// TIA Portal V19 export
FUNCTION "SCALING_PARAMETERS" : Void   // FC4, LAD
{ S7_Optimized_Access := 'TRUE' }
// stored: SetENOAutomatically false
BEGIN

REGION Network 1: PH_SCALE
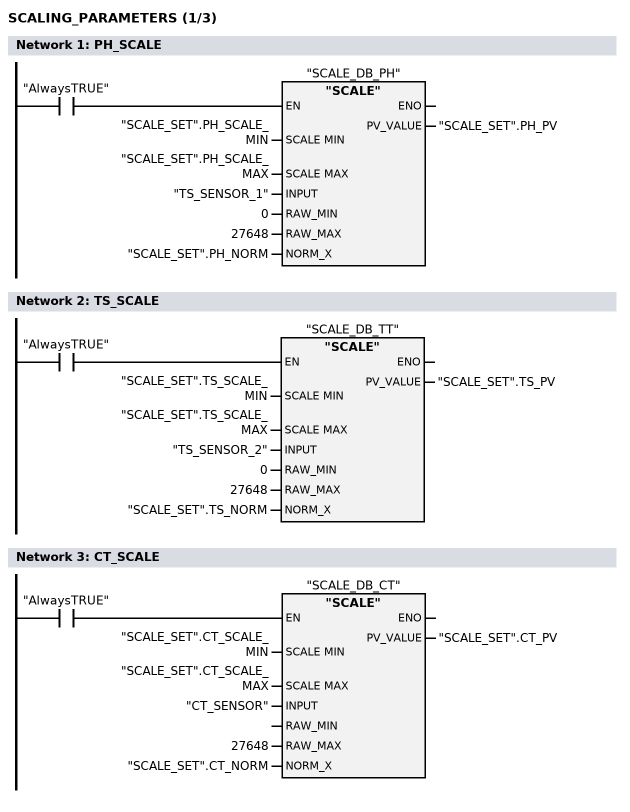
   RUNG wire#powerrail
      Contact( "AlwaysTRUE" )
      "SCALE_DB_PH"("SCALE MIN" := "SCALE_SET".PH_SCALE_MIN, "SCALE MAX" := "SCALE_SET".PH_SCALE_MAX, INPUT := "TS_SENSOR_1", RAW_MIN := 0, RAW_MAX := 27648, NORM_X := "SCALE_SET".PH_NORM, PV_VALUE => "SCALE_SET".PH_PV)
   END_RUNG
   // the same network as SCL:
   IF "AlwaysTRUE" THEN
       "SCALE_DB_PH"("SCALE MIN" := "SCALE_SET".PH_SCALE_MIN,   // "SCALE"
                     "SCALE MAX" := "SCALE_SET".PH_SCALE_MAX,
                     INPUT := "TS_SENSOR_1",
                     RAW_MIN := 0,
                     RAW_MAX := 27648,
                     NORM_X := "SCALE_SET".PH_NORM,
                     PV_VALUE => "SCALE_SET".PH_PV);
   END_IF;
END_REGION

REGION Network 2: TS_SCALE
   RUNG wire#powerrail
      Contact( "AlwaysTRUE" )
      "SCALE_DB_TT"("SCALE MIN" := "SCALE_SET".TS_SCALE_MIN, "SCALE MAX" := "SCALE_SET".TS_SCALE_MAX, INPUT := "TS_SENSOR_2", RAW_MIN := 0, RAW_MAX := 27648, NORM_X := "SCALE_SET".TS_NORM, PV_VALUE => "SCALE_SET".TS_PV)
   END_RUNG
   // the same network as SCL:
   IF "AlwaysTRUE" THEN
       "SCALE_DB_TT"("SCALE MIN" := "SCALE_SET".TS_SCALE_MIN,   // "SCALE"
                     "SCALE MAX" := "SCALE_SET".TS_SCALE_MAX,
                     INPUT := "TS_SENSOR_2",
                     RAW_MIN := 0,
                     RAW_MAX := 27648,
                     NORM_X := "SCALE_SET".TS_NORM,
                     PV_VALUE => "SCALE_SET".TS_PV);
   END_IF;
END_REGION

REGION Network 3: CT_SCALE
   RUNG wire#powerrail
      Contact( "AlwaysTRUE" )
      "SCALE_DB_CT"("SCALE MIN" := "SCALE_SET".CT_SCALE_MIN, "SCALE MAX" := "SCALE_SET".CT_SCALE_MAX, INPUT := "CT_SENSOR", RAW_MIN :=, RAW_MAX := 27648, NORM_X := "SCALE_SET".CT_NORM, PV_VALUE => "SCALE_SET".CT_PV)
   END_RUNG
   // the same network as SCL:
   IF "AlwaysTRUE" THEN
       "SCALE_DB_CT"("SCALE MIN" := "SCALE_SET".CT_SCALE_MIN,   // "SCALE"
                     "SCALE MAX" := "SCALE_SET".CT_SCALE_MAX,
                     INPUT := "CT_SENSOR",
                     RAW_MAX := 27648,
                     NORM_X := "SCALE_SET".CT_NORM,
                     PV_VALUE => "SCALE_SET".CT_PV);
   END_IF;
END_REGION

REGION Network 4: SET_PUMP_SPEED
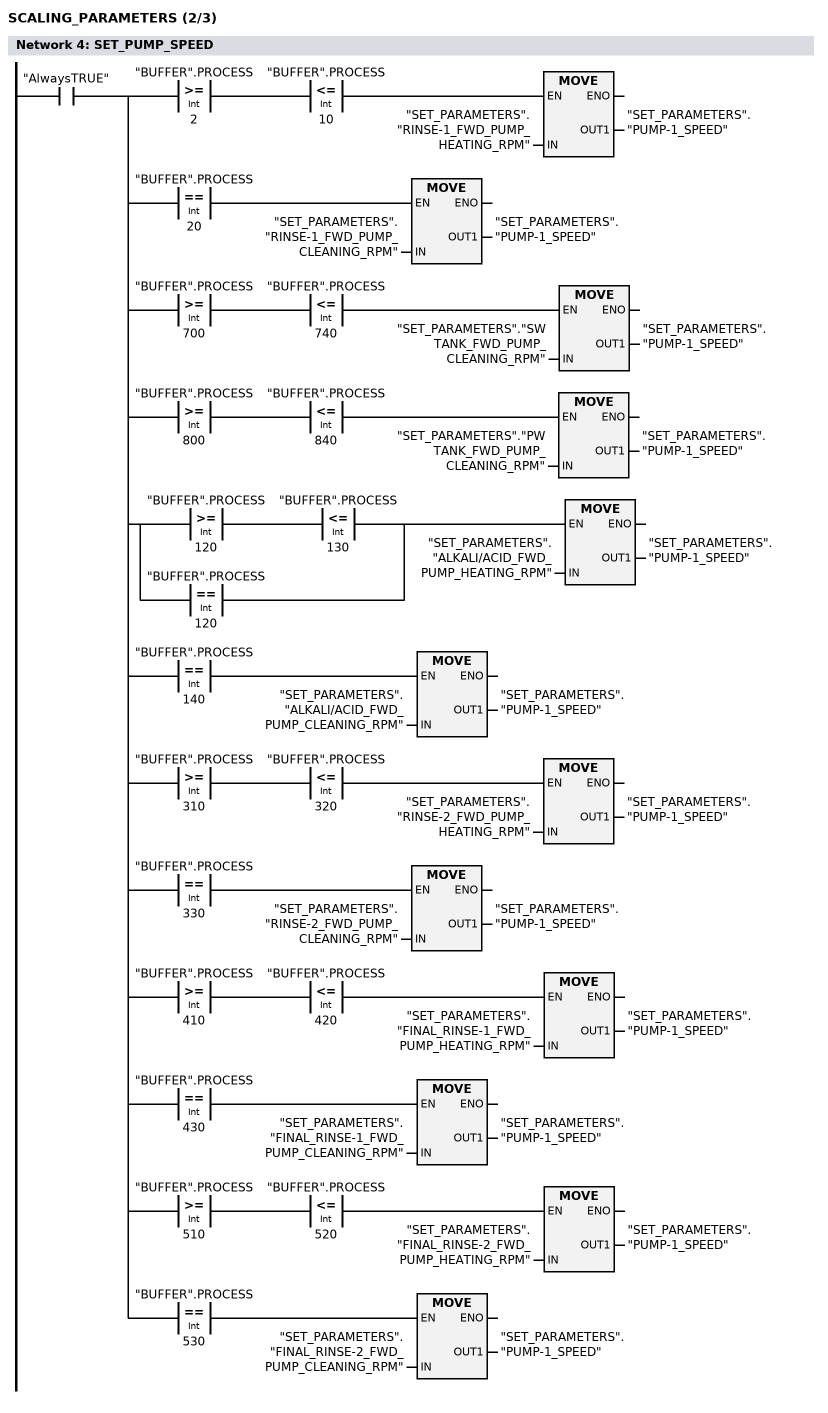
   RUNG wire#powerrail
      Contact( "AlwaysTRUE" )
      wire#w1
      { S7_Templates := "SrcType := Int" } GE_Contact(in1 := "BUFFER".PROCESS, in2 := 2)
      { S7_Templates := "SrcType := Int" } LE_Contact(in1 := "BUFFER".PROCESS, in2 := 10)
      Move(in := "SET_PARAMETERS"."RINSE-1_FWD_PUMP_HEATING_RPM", out1 => "SET_PARAMETERS"."PUMP-1_SPEED")
   END_RUNG
   RUNG wire#w1
      { S7_Templates := "SrcType := Int" } EQ_Contact(in1 := "BUFFER".PROCESS, in2 := 20)
      Move(in := "SET_PARAMETERS"."RINSE-1_FWD_PUMP_CLEANING_RPM", out1 => "SET_PARAMETERS"."PUMP-1_SPEED")
   END_RUNG
   RUNG wire#w1
      { S7_Templates := "SrcType := Int" } GE_Contact(in1 := "BUFFER".PROCESS, in2 := 700)
      { S7_Templates := "SrcType := Int" } LE_Contact(in1 := "BUFFER".PROCESS, in2 := 740)
      Move(in := "SET_PARAMETERS"."SW TANK_FWD_PUMP_CLEANING_RPM", out1 => "SET_PARAMETERS"."PUMP-1_SPEED")
   END_RUNG
   RUNG wire#w1
      { S7_Templates := "SrcType := Int" } GE_Contact(in1 := "BUFFER".PROCESS, in2 := 800)
      { S7_Templates := "SrcType := Int" } LE_Contact(in1 := "BUFFER".PROCESS, in2 := 840)
      Move(in := "SET_PARAMETERS"."PW TANK_FWD_PUMP_CLEANING_RPM", out1 => "SET_PARAMETERS"."PUMP-1_SPEED")
   END_RUNG
   RUNG wire#w1
      { S7_Templates := "SrcType := Int" } GE_Contact(in1 := "BUFFER".PROCESS, in2 := 120)
      { S7_Templates := "SrcType := Int" } LE_Contact(in1 := "BUFFER".PROCESS, in2 := 130)
      wire#w2
      Move(in := "SET_PARAMETERS"."ALKALI/ACID_FWD_PUMP_HEATING_RPM", out1 => "SET_PARAMETERS"."PUMP-1_SPEED")
   END_RUNG
   RUNG wire#w1
      { S7_Templates := "SrcType := Int" } EQ_Contact(in1 := "BUFFER".PROCESS, in2 := 120)
   END_RUNG wire#w2
   RUNG wire#w1
      { S7_Templates := "SrcType := Int" } EQ_Contact(in1 := "BUFFER".PROCESS, in2 := 140)
      Move(in := "SET_PARAMETERS"."ALKALI/ACID_FWD_PUMP_CLEANING_RPM", out1 => "SET_PARAMETERS"."PUMP-1_SPEED")
   END_RUNG
   RUNG wire#w1
      { S7_Templates := "SrcType := Int" } GE_Contact(in1 := "BUFFER".PROCESS, in2 := 310)
      { S7_Templates := "SrcType := Int" } LE_Contact(in1 := "BUFFER".PROCESS, in2 := 320)
      Move(in := "SET_PARAMETERS"."RINSE-2_FWD_PUMP_HEATING_RPM", out1 => "SET_PARAMETERS"."PUMP-1_SPEED")
   END_RUNG
   RUNG wire#w1
      { S7_Templates := "SrcType := Int" } EQ_Contact(in1 := "BUFFER".PROCESS, in2 := 330)
      Move(in := "SET_PARAMETERS"."RINSE-2_FWD_PUMP_CLEANING_RPM", out1 => "SET_PARAMETERS"."PUMP-1_SPEED")
   END_RUNG
   RUNG wire#w1
      { S7_Templates := "SrcType := Int" } GE_Contact(in1 := "BUFFER".PROCESS, in2 := 410)
      { S7_Templates := "SrcType := Int" } LE_Contact(in1 := "BUFFER".PROCESS, in2 := 420)
      Move(in := "SET_PARAMETERS"."FINAL_RINSE-1_FWD_PUMP_HEATING_RPM", out1 => "SET_PARAMETERS"."PUMP-1_SPEED")
   END_RUNG
   RUNG wire#w1
      { S7_Templates := "SrcType := Int" } EQ_Contact(in1 := "BUFFER".PROCESS, in2 := 430)
      Move(in := "SET_PARAMETERS"."FINAL_RINSE-1_FWD_PUMP_CLEANING_RPM", out1 => "SET_PARAMETERS"."PUMP-1_SPEED")
   END_RUNG
   RUNG wire#w1
      { S7_Templates := "SrcType := Int" } GE_Contact(in1 := "BUFFER".PROCESS, in2 := 510)
      { S7_Templates := "SrcType := Int" } LE_Contact(in1 := "BUFFER".PROCESS, in2 := 520)
      Move(in := "SET_PARAMETERS"."FINAL_RINSE-2_FWD_PUMP_HEATING_RPM", out1 => "SET_PARAMETERS"."PUMP-1_SPEED")
   END_RUNG
   RUNG wire#w1
      { S7_Templates := "SrcType := Int" } EQ_Contact(in1 := "BUFFER".PROCESS, in2 := 530)
      Move(in := "SET_PARAMETERS"."FINAL_RINSE-2_FWD_PUMP_CLEANING_RPM", out1 => "SET_PARAMETERS"."PUMP-1_SPEED")
   END_RUNG
   // the same network as SCL:
   IF "AlwaysTRUE" AND ("BUFFER".PROCESS >= 2) AND ("BUFFER".PROCESS <= 10) THEN
       "SET_PARAMETERS"."PUMP-1_SPEED" := "SET_PARAMETERS"."RINSE-1_FWD_PUMP_HEATING_RPM";
   END_IF;
   IF "AlwaysTRUE" AND ("BUFFER".PROCESS = 20) THEN
       "SET_PARAMETERS"."PUMP-1_SPEED" := "SET_PARAMETERS"."RINSE-1_FWD_PUMP_CLEANING_RPM";
   END_IF;
   IF "AlwaysTRUE" AND ("BUFFER".PROCESS >= 700) AND ("BUFFER".PROCESS <= 740) THEN
       "SET_PARAMETERS"."PUMP-1_SPEED" := "SET_PARAMETERS"."SW TANK_FWD_PUMP_CLEANING_RPM";
   END_IF;
   IF "AlwaysTRUE" AND ("BUFFER".PROCESS >= 800) AND ("BUFFER".PROCESS <= 840) THEN
       "SET_PARAMETERS"."PUMP-1_SPEED" := "SET_PARAMETERS"."PW TANK_FWD_PUMP_CLEANING_RPM";
   END_IF;
   IF "AlwaysTRUE" AND ((("BUFFER".PROCESS >= 120) AND ("BUFFER".PROCESS <= 130)) OR ("BUFFER".PROCESS = 120)) THEN
       "SET_PARAMETERS"."PUMP-1_SPEED" := "SET_PARAMETERS"."ALKALI/ACID_FWD_PUMP_HEATING_RPM";
   END_IF;
   IF "AlwaysTRUE" AND ("BUFFER".PROCESS = 140) THEN
       "SET_PARAMETERS"."PUMP-1_SPEED" := "SET_PARAMETERS"."ALKALI/ACID_FWD_PUMP_CLEANING_RPM";
   END_IF;
   IF "AlwaysTRUE" AND ("BUFFER".PROCESS >= 310) AND ("BUFFER".PROCESS <= 320) THEN
       "SET_PARAMETERS"."PUMP-1_SPEED" := "SET_PARAMETERS"."RINSE-2_FWD_PUMP_HEATING_RPM";
   END_IF;
   IF "AlwaysTRUE" AND ("BUFFER".PROCESS = 330) THEN
       "SET_PARAMETERS"."PUMP-1_SPEED" := "SET_PARAMETERS"."RINSE-2_FWD_PUMP_CLEANING_RPM";
   END_IF;
   IF "AlwaysTRUE" AND ("BUFFER".PROCESS >= 410) AND ("BUFFER".PROCESS <= 420) THEN
       "SET_PARAMETERS"."PUMP-1_SPEED" := "SET_PARAMETERS"."FINAL_RINSE-1_FWD_PUMP_HEATING_RPM";
   END_IF;
   IF "AlwaysTRUE" AND ("BUFFER".PROCESS = 430) THEN
       "SET_PARAMETERS"."PUMP-1_SPEED" := "SET_PARAMETERS"."FINAL_RINSE-1_FWD_PUMP_CLEANING_RPM";
   END_IF;
   IF "AlwaysTRUE" AND ("BUFFER".PROCESS >= 510) AND ("BUFFER".PROCESS <= 520) THEN
       "SET_PARAMETERS"."PUMP-1_SPEED" := "SET_PARAMETERS"."FINAL_RINSE-2_FWD_PUMP_HEATING_RPM";
   END_IF;
   IF "AlwaysTRUE" AND ("BUFFER".PROCESS = 530) THEN
       "SET_PARAMETERS"."PUMP-1_SPEED" := "SET_PARAMETERS"."FINAL_RINSE-2_FWD_PUMP_CLEANING_RPM";
   END_IF;
END_REGION

REGION Network 5: PUMP-1 SPEED
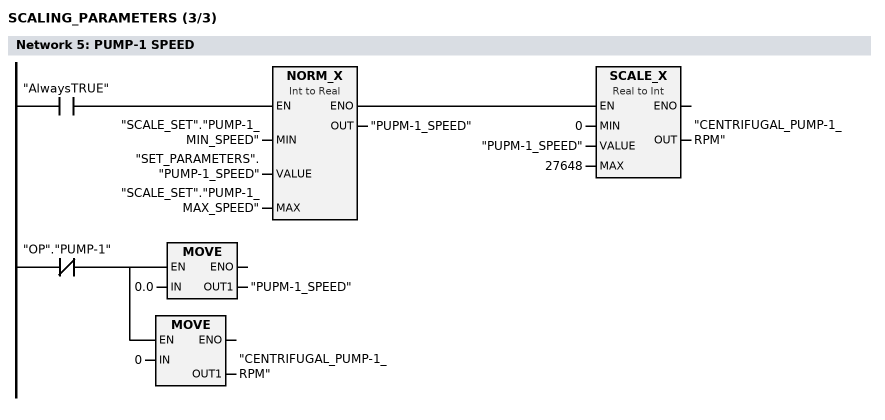
   RUNG wire#powerrail
      Contact( "AlwaysTRUE" )
      { S7_Templates := "[SrcType := Int, DestType := Real]" } Normalize(min := "SCALE_SET"."PUMP-1_MIN_SPEED", value := "SET_PARAMETERS"."PUMP-1_SPEED", max := "SCALE_SET"."PUMP-1_MAX_SPEED", out => "PUPM-1_SPEED")
      { S7_Templates := "[SrcType := Real, DestType := Int]" } Scale(min := 0, value := "PUPM-1_SPEED", max := 27648, out => "CENTRIFUGAL_PUMP-1_RPM")
   END_RUNG
   RUNG wire#powerrail
      I_Contact( "OP"."PUMP-1" )
      wire#w1
      Move(in := 0.0, out1 => "PUPM-1_SPEED")
   END_RUNG
   RUNG wire#w1
      Move(in := 0, out1 => "CENTRIFUGAL_PUMP-1_RPM")
   END_RUNG
   // the same network as SCL:
   IF "AlwaysTRUE" THEN
       "PUPM-1_SPEED" := NORM_X(MIN := "SCALE_SET"."PUMP-1_MIN_SPEED", VALUE := "SET_PARAMETERS"."PUMP-1_SPEED", MAX := "SCALE_SET"."PUMP-1_MAX_SPEED");
       "CENTRIFUGAL_PUMP-1_RPM" := SCALE_X(MIN := 0, VALUE := "PUPM-1_SPEED", MAX := 27648);
   END_IF;
   IF NOT "OP"."PUMP-1" THEN
       "PUPM-1_SPEED" := 0.0;
       "CENTRIFUGAL_PUMP-1_RPM" := 0;
   END_IF;
END_REGION
END_FUNCTION
